// TIA Portal V17 export
// export: Created 2024-06-14T09:53:10.713342Z, ExportSetting WithDefaults, DisplayName Totally Integrated Automation Portal, DisplayVersion V17, DisplayName TIA Portal Openness, DisplayVersion V17, DisplayName TIA Portal Version Control Interface, DisplayVersion V17, DisplayName Simotion SCOUT TIA, DisplayVersion 5.4.3.0, DisplayName SINAMICS Startdrive Advanced, DisplayVersion V17 SP1 Update 1, DisplayName SINAMICS Startdrive G110M, G120, G120C, G120D, G120P, G115D, DisplayVersion V17 SP1 Update 1, DisplayName SINAMICS Startdrive G130, G150, S120, S150, SINAMICS MV, S210, DisplayVersion V17 SP1 Update 1, DisplayName STEP 7 Professional, DisplayVersion V17, DisplayName STEP 7 Safety, DisplayVersion V17, DisplayName WinCC Professional, DisplayVersion V17
DATA_BLOCK "Check_scale_LPG_DB"   // DB47
VERSION : 0.1
// stored: AutoNumber true, DBAccessibleFromOPCUA true, InstanceOfName Check_scale_LPG, InstanceOfType FB
"Check_scale_LPG"
   // VAR_INPUT
   //    Stopper_sesnor : Bool;
   //    Cylinder_presence : Bool;
   //    Pass_line_jammer : Bool;
   //    Down_line_jammer : Bool;
   //    Start_cycle : Bool;
   //    Reset_Cycle : Bool;
   //    Result : Int;
   //    Pusher : Bool;
   //    all_fill_done : Bool;
   //    xResult : Bool;
   // END_VAR
   // VAR_OUTPUT
   //    Stopper : Bool;
   //    LiftTable : Bool;
   //    Start_Check_Scale : Bool;
   //    Divider : Bool;
   //    Reset : Bool;
   //    CYCLE_ONE : Bool;
   // END_VAR
   // VAR
   //    Check_Scale_Started : Bool;
   //    Lift_Table { S7_SetPoint := 'True'} : TON_TIME;
   //    PASS : Bool;
   //    FAIL : Bool;
   //    LIFT_down { S7_SetPoint := 'True'} : TON_TIME;
   //    Temp_1 : Int;
   //    p_trig : Array[0..10] of Bool;
   // END_VAR
   // VAR RETAIN
   //    Stopper_count { S7_SetPoint := 'True'} : CTU_INT;
   // END_VAR
   // VAR
   //    counter_reset : Bool;
   //    Scale { S7_SetPoint := 'True'} : TON_TIME;
   //    Pusher_reset { S7_SetPoint := 'True'} : TON_TIME;
   //    datasend { ExternalAccessible := 'False'; ExternalVisible := 'False'; ExternalWritable := 'False'} : Bool;
   //    fb_Fifo_Instance { S7_SetPoint := 'True'} : "fb_Fifo";
   //    idx7 : Int;
   //    fb_Compress_Instance { S7_SetPoint := 'True'} : "fb_Compress";
   //    jammer_on { S7_SetPoint := 'True'} : TON_TIME;
   //    jammer : Bool;
   //    pusher_enable : Bool;
   //    Scale_done : Bool;
   // END_VAR
   // VAR RETAIN
   //    Lift_Table_UP { S7_SetPoint := 'True'} : CTU_INT;
   // END_VAR
   // VAR
   //    fb_Fifo_Instance_1 { S7_SetPoint := 'True'} : "fb_Fifo";
   //    fb_Compress_Instance_1 { S7_SetPoint := 'True'} : "fb_Compress";
   //    timer_1 { S7_SetPoint := 'True'} : TON_TIME;
   // END_VAR
BEGIN
END_DATA_BLOCK
